FUNCTION CableVelocityToMotorAngularVelocity : LREAL
VAR_INPUT
	cable_velocity : LREAL;
END_VAR
VAR_OUTPUT
	motor_velocity : LREAL;
END_VAR
VAR
END_VAR

motor_velocity := cable_velocity;

END_FUNCTION

(* stored: Version 1.1.0.1, ProductVersion 3.1.4024.11
   POU CableVelocityToMotorAngularVelocity: Id {3d32bdbe-11b5-4ae5-bf28-72298521e5c1}, SpecialFunc None *)
